// Struckig
// Copyright (C) 2022 Stefan Besler

// This program is free software: you can redistribute it and/or modify
// it under the terms of the GNU General Public License as published by
// the Free Software Foundation, either version 3 of the License, or
// (at your option) any later version.

// This program is distributed in the hope that it will be useful,
// but WITHOUT ANY WARRANTY; without even the implied warranty of
// MERCHANTABILITY or FITNESS FOR A PARTICULAR PURPOSE.  See the
// GNU General Public License for more details.
//
// You should have received a copy of the GNU General Public License
// along with THIS PROGRAM.  IF NOT, see <http://www.gnu.org/licenses/>.
{attribute 'qualified_only'}
{attribute 'strict'}
/// Defines how multiple DoFs are synchronized to a common trajectory timing.
/// This setting is evaluated together with per-axis overrides (`PerDofSynchronization`)
/// in [Otg](xref:Struckig.Otg).
TYPE SynchronizationType :
(
  Undefined, //< Use global/default configuration.
  TimeSync, //< Always synchronize the DoFs to reach the target at the same time (Default)
  TimeIfNecessarySync, //< Synchronize only when necessary (e.g. for non-zero target velocity or acceleration)
  Phase,  //< Phase synchronize the DoFs when this is possible, else fallback to "Time" strategy. Phase synchronization will result a straight-line trajectory
    // PhaseOnly, //< Always phase synchronize the DoFs (even when this is not time-optimal), else returns "ErrorNoPhaseSynchronization". Ruckig will then guarantee a straight-line trajectory
  None //< Calculate every DoF independently
);
END_TYPE

(* stored: Version 1.1.0.1
   DUT SynchronizationType: Id {c2f32290-f62f-4354-9b4e-71d37ff75e54} *)
